      CALL #FW_APW_Oeb_PG
      (  Idx                         := 4 ,
         Niv_Frg                     := #akt_Niv_ZS_AS ,
         Frg_Aus                     := #PW_all_Frg_Aus ,
         Frg_Ein                     := #PW_all_Frg_Ein ,
         DF_Skal                     := 30.0 ,
         IEC_Image                   := "DB_IEC_PW_Image".FW_APW_Oeb_PG ,
         PW_Meld                     := "DB118_PW_Meld".FW_APW_Oeb_PG ,
         PW_Bef                      := "DB119_PW_Bef".FW_APW_Oeb_PG ,
         AS_Zyk                      := #PW_all_Frg_AS_zyk ,
         ZS_Zyk                      := #PW_all_Frg_ZS_zyk ,
         RM_Frg_Ein                  := #PW_all_RM_Frg_Ein ,
         RM_Frg_TeilAus              := #PW_all_RM_Frg_TeilAus ,
         RM_Frg_Aus                  := #PW_all_RM_Frg_Aus
      );

      CALL #FW_APW_Oeb_LW
      (  Idx                         := 5 ,
         Niv_Frg                     := #akt_Niv_ZS_AS ,
         Frg_Aus                     := #PW_all_Frg_Aus ,
         Frg_Ein                     := #PW_all_Frg_Ein ,
         Sperre_ext                  := 0 ,
         DF_Skal                     := 30.0 ,
         IEC_Image                   := "DB_IEC_PW_Image".FW_APW_Oeb_LW ,
         PW_Meld                     := "DB118_PW_Meld".FW_APW_Oeb_LW ,
         PW_Bef                      := "DB119_PW_Bef".FW_APW_Oeb_LW ,
         AS_Zyk                      := #PW_all_Frg_AS_zyk ,
         ZS_Zyk                      := #PW_all_Frg_ZS_zyk ,
         RM_Frg_Ein                  := #PW_all_RM_Frg_Ein ,
         RM_Frg_TeilAus              := #PW_all_RM_Frg_TeilAus ,
         RM_Frg_Aus                  := #PW_all_RM_Frg_Aus
      );

      CALL #FW_APW_GeD_WG
      (  Idx                         := 6 ,
         Niv_Frg                     := #akt_Niv_ZS_AS ,
         Frg_Aus                     := #PW_all_Frg_Aus ,
         Frg_Ein                     := #PW_all_Frg_Ein ,
         IEC_Image                   := "DB_IEC_PW_Image".FW_APW_GeD_WG ,
         PW_Meld                     := "DB118_PW_Meld".FW_APW_GeD_WG ,
         PW_Bef                      := "DB119_PW_Bef".FW_APW_GeD_WG ,
         AS_Zyk                      := #PW_all_Frg_AS_zyk ,
         ZS_Zyk                      := #PW_all_Frg_ZS_zyk ,
         RM_Frg_Ein                  := #PW_all_RM_Frg_Ein ,
         RM_Frg_TeilAus              := #PW_all_RM_Frg_TeilAus ,
         RM_Frg_Aus                  := #PW_all_RM_Frg_Aus
      );

      CALL #FW_APW_GeD_AA
      (  Idx                         := 7 ,
         Niv_Frg                     := #akt_Niv_ZS_AS ,
         Frg_Aus                     := #PW_all_Frg_Aus ,
         Frg_Ein                     := #PW_all_Frg_Ein ,
         IEC_Image                   := "DB_IEC_PW_Image".FW_APW_GeD_AA ,
         PW_Meld                     := "DB118_PW_Meld".FW_APW_GeD_AA ,
         PW_Bef                      := "DB119_PW_Bef".FW_APW_GeD_AA ,
         AS_Zyk                      := #PW_all_Frg_AS_zyk ,
         ZS_Zyk                      := #PW_all_Frg_ZS_zyk ,
         RM_Frg_Ein                  := #PW_all_RM_Frg_Ein ,
         RM_Frg_TeilAus              := #PW_all_RM_Frg_TeilAus ,
         RM_Frg_Aus                  := #PW_all_RM_Frg_Aus
      );

      U "DB118_PW_Meld".FW_APW_WaD.Status.FWA_Betrieb;
      UN #FW_APW_WaD.Sperre_ext;
      S #FW_APW_WeD.Sperre_ext;
      S #FW_APW_NiD.Sperre_ext;

      UN "DB118_PW_Meld".FW_APW_WaD.Status.FWA_Betrieb;
      UN #FW_APW_WaD.Sperre_ext;
      R #FW_APW_WeD.Sperre_ext;
      R #FW_APW_NiD.Sperre_ext;

      CALL #FW_APW_WaD
      (  Idx                         := 8 ,
         Niv_Frg                     := #akt_Niv_ZS_AS ,
         Frg_Aus                     := #PW_all_Frg_Aus ,
         Frg_Ein                     := #PW_all_Frg_Ein ,
         IEC_Image                   := "DB_IEC_PW_Image".FW_APW_WaD ,
         PW_Meld                     := "DB118_PW_Meld".FW_APW_WaD ,
         PW_Bef                      := "DB119_PW_Bef".FW_APW_WaD ,
         AS_Zyk                      := #PW_all_Frg_AS_zyk ,
         ZS_Zyk                      := #PW_all_Frg_ZS_zyk ,
         RM_Frg_Ein                  := #PW_all_RM_Frg_Ein ,
         RM_Frg_TeilAus              := #PW_all_RM_Frg_TeilAus ,
         RM_Frg_Aus                  := #PW_all_RM_Frg_Aus
      );

      U "DB118_PW_Meld".FW_APW_WeD.Status.FWA_Betrieb;
      UN #FW_APW_WeD.Sperre_ext;
      S #FW_APW_WaD.Sperre_ext;
      S #FW_APW_NiD.Sperre_ext;

      UN "DB118_PW_Meld".FW_APW_WeD.Status.FWA_Betrieb;
      UN #FW_APW_WeD.Sperre_ext;
      R #FW_APW_WaD.Sperre_ext;
      R #FW_APW_NiD.Sperre_ext;


      CALL #FW_APW_WeD
      (  Idx                         := 9 ,
         Niv_Frg                     := #akt_Niv_ZS_AS ,
         Frg_Aus                     := #PW_all_Frg_Aus ,
         Frg_Ein                     := #PW_all_Frg_Ein ,
         IEC_Image                   := "DB_IEC_PW_Image".FW_APW_WeD ,
         PW_Meld                     := "DB118_PW_Meld".FW_APW_WeD ,
         PW_Bef                      := "DB119_PW_Bef".FW_APW_WeD ,
         AS_Zyk                      := #PW_all_Frg_AS_zyk ,
         ZS_Zyk                      := #PW_all_Frg_ZS_zyk ,
         RM_Frg_Ein                  := #PW_all_RM_Frg_Ein ,
         RM_Frg_TeilAus              := #PW_all_RM_Frg_TeilAus ,
         RM_Frg_Aus                  := #PW_all_RM_Frg_Aus
      );

      U "DB118_PW_Meld".FW_APW_NiD.Status.FWA_Betrieb;
      UN #FW_APW_NiD.Sperre_ext;
      S #FW_APW_WeD.Sperre_ext;
      S #FW_APW_WaD.Sperre_ext;

      UN "DB118_PW_Meld".FW_APW_NiD.Status.FWA_Betrieb;
      UN #FW_APW_NiD.Sperre_ext;
      R #FW_APW_WeD.Sperre_ext;
      R #FW_APW_WaD.Sperre_ext;

      CALL #FW_APW_NiD
      (  Idx                         := 10 ,
         Niv_Frg                     := #akt_Niv_ZS_AS ,
         Frg_Aus                     := #PW_all_Frg_Aus ,
         Frg_Ein                     := #PW_all_Frg_Ein ,
         IEC_Image                   := "DB_IEC_PW_Image".FW_APW_NiD ,
         PW_Meld                     := "DB118_PW_Meld".FW_APW_NiD ,
         PW_Bef                      := "DB119_PW_Bef".FW_APW_NiD ,
         AS_Zyk                      := #PW_all_Frg_AS_zyk ,
         ZS_Zyk                      := #PW_all_Frg_ZS_zyk ,
         RM_Frg_Ein                  := #PW_all_RM_Frg_Ein ,
         RM_Frg_TeilAus              := #PW_all_RM_Frg_TeilAus ,
         RM_Frg_Aus                  := #PW_all_RM_Frg_Aus
      );

      CALL #FW_APW_LoS
      (  Idx                         := 11 ,
         Niv_Frg                     := #akt_Niv_ZS_AS ,
         Frg_Aus                     := #PW_all_Frg_Aus ,
         Frg_Ein                     := #PW_all_Frg_Ein ,
         IEC_Image                   := "DB_IEC_PW_Image".FW_APW_LoS ,
         PW_Meld                     := "DB118_PW_Meld".FW_APW_LoS ,
         PW_Bef                      := "DB119_PW_Bef".FW_APW_LoS ,
         AS_Zyk                      := #PW_all_Frg_AS_zyk ,
         ZS_Zyk                      := #PW_all_Frg_ZS_zyk ,
         RM_Frg_Ein                  := #PW_all_RM_Frg_Ein ,
         RM_Frg_TeilAus              := #PW_all_RM_Frg_TeilAus ,
         RM_Frg_Aus                  := #PW_all_RM_Frg_Aus
      );

      CALL #FW_APW_Oeb_Ge
      (  Idx                         := 12 ,
         Niv_Frg                     := #akt_Niv_ZS_AS ,
         Frg_Aus                     := #PW_all_Frg_Aus ,
         Frg_Ein                     := #PW_all_Frg_Ein ,
         DF_Skal                     := 20.0 ,
         IEC_Image                   := "DB_IEC_PW_Image".FW_APW_Oeb_Ge ,
         PW_Meld                     := "DB118_PW_Meld".FW_APW_Oeb_Ge ,
         PW_Bef                      := "DB119_PW_Bef".FW_APW_Oeb_Ge ,
         AS_Zyk                      := #PW_all_Frg_AS_zyk ,
         ZS_Zyk                      := #PW_all_Frg_ZS_zyk ,
         RM_Frg_Ein                  := #PW_all_RM_Frg_Ein ,
         RM_Frg_TeilAus              := #PW_all_RM_Frg_TeilAus ,
         RM_Frg_Aus                  := #PW_all_RM_Frg_Aus
      );

      CALL #FW_APW_BuH
      (  Idx                         := 13 ,
         Niv_Frg                     := #akt_Niv_ZS_AS ,
         Frg_Aus                     := #PW_all_Frg_Aus ,
         Frg_Ein                     := #PW_all_Frg_Ein ,
         IEC_Image                   := "DB_IEC_PW_Image".FW_APW_BuH ,
         PW_Meld                     := "DB118_PW_Meld".FW_APW_BuH ,
         PW_Bef                      := "DB119_PW_Bef".FW_APW_BuH ,
         AS_Zyk                      := #PW_all_Frg_AS_zyk ,
         ZS_Zyk                      := #PW_all_Frg_ZS_zyk ,
         RM_Frg_Ein                  := #PW_all_RM_Frg_Ein ,
         RM_Frg_TeilAus              := #PW_all_RM_Frg_TeilAus ,
         RM_Frg_Aus                  := #PW_all_RM_Frg_Aus
      );

      CALL #FW_APW_BrR_TS
      (  Idx                         := 14 ,
         Niv_Frg                     := #akt_Niv_ZS_AS ,
         Frg_Aus                     := #PW_all_Frg_Aus ,
         Frg_Ein                     := #PW_all_Frg_Ein ,
         IEC_Image                   := "DB_IEC_PW_Image".FW_APW_BrR_TS ,
         PW_Meld                     := "DB118_PW_Meld".FW_APW_BrR_TS ,
         PW_Bef                      := "DB119_PW_Bef".FW_APW_BrR_TS ,
         AS_Zyk                      := #PW_all_Frg_AS_zyk ,
         ZS_Zyk                      := #PW_all_Frg_ZS_zyk ,
         RM_Frg_Ein                  := #PW_all_RM_Frg_Ein ,
         RM_Frg_TeilAus              := #PW_all_RM_Frg_TeilAus ,
         RM_Frg_Aus                  := #PW_all_RM_Frg_Aus
      );

NETWORK
TITLE = Steuerung Zulauf/Freigabe Pumpwerke - Status - alle Freigaben
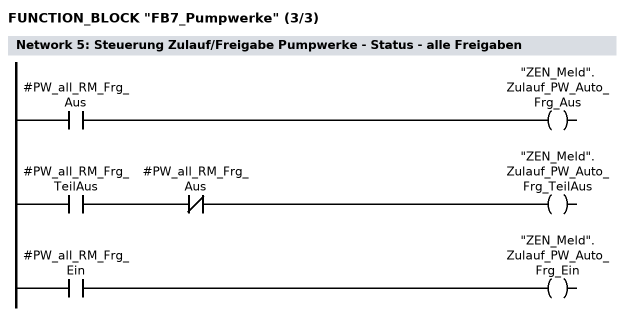

      U #PW_all_RM_Frg_Aus;
      = "ZEN_Meld".Zulauf_PW_Auto_Frg_Aus;
      U #PW_all_RM_Frg_TeilAus;
      UN #PW_all_RM_Frg_Aus;
      = "ZEN_Meld".Zulauf_PW_Auto_Frg_TeilAus;
      U #PW_all_RM_Frg_Ein;
      = "ZEN_Meld".Zulauf_PW_Auto_Frg_Ein;


END_FUNCTION_BLOCK

FUNCTION_BLOCK "FB8_Leitstelle"
{ S7_Optimized_Access := 'TRUE' }
VERSION : 0.1
   VAR_TEMP
      BB_G1_SS : Bool;
      BB_G2_SS : Bool;
      BB_G3_SS : Bool;
      retval : Int;
   END_VAR


BEGIN
NETWORK
TITLE = Sammelmeldung an Leitstelle - Gebläse 1 Störung
      U "DB104_Antriebe_Meld".BB_G1.Status.BB_SS;
      O "DB104_Antriebe_Meld".BB_G1.Stoerung.St_Kom_DP;
      = #BB_G1_SS;
      U "DB104_Antriebe_Meld".BB_G2.Status.BB_SS;
      O "DB104_Antriebe_Meld".BB_G2.Stoerung.St_Kom_DP;
      = #BB_G2_SS;
      U "DB104_Antriebe_Meld".BB_G3.Status.BB_SS;
      O "DB104_Antriebe_Meld".BB_G3.Stoerung.St_Kom_DP;
      = #BB_G3_SS;

//Gebläse 1 Störung
      U #BB_G1_SS;
      = "ZEN_Meld".IEC_Meld_LS_001;
//Gebläse 2 Störung
      U #BB_G2_SS;
      = "ZEN_Meld".IEC_Meld_LS_002;
//Gebläse 3 Störung
      U #BB_G3_SS;
      = "ZEN_Meld".IEC_Meld_LS_003;

//Belebungsbecken 1 Rezipumpe 1 Störung
      U "DB104_Antriebe_Meld".BB1_RZP1.Status.BB_SS;
      = "ZEN_Meld".IEC_Meld_LS_004;

//Belebungsbecken 1 Rezipumpe 2 Störung
      U "DB104_Antriebe_Meld".BB1_RZP2.Status.BB_SS;
      = "ZEN_Meld".IEC_Meld_LS_005;

//Belebungsbecken 1 Überschussschlammpumpe Störung
      U "DB104_Antriebe_Meld".BB1_UeSP.Status.BB_SS;
      = "ZEN_Meld".IEC_Meld_LS_006;

//Belebungsbecken 1 Ablaufschieber Störung
      U "DB104_Antriebe_Meld".BB1_AS1.Status.BB_SS;
      O "DB104_Antriebe_Meld".BB1_AS2.Status.BB_SS;
      = "ZEN_Meld".IEC_Meld_LS_007;

//Belebungsbecken 1 Schlammrückführung Störung
      U "DB104_Antriebe_Meld".BB1_SR1.Status.BB_SS;
      O "DB104_Antriebe_Meld".BB1_SR2.Status.BB_SS;
      = "ZEN_Meld".IEC_Meld_LS_008;

//Belebungsbecken 2 Rezipumpe 1 Störung
      U "DB104_Antriebe_Meld".BB2_RZP1.Status.BB_SS;
      = "ZEN_Meld".IEC_Meld_LS_009;

//Belebungsbecken 2 Rezipumpe 2 Störung
      U "DB104_Antriebe_Meld".BB2_RZP2.Status.BB_SS;
      = "ZEN_Meld".IEC_Meld_LS_010;

//Belebungsbecken 2 Überschussschlammpumpe Störung
      U "DB104_Antriebe_Meld".BB2_UeSP.Status.BB_SS;
      = "ZEN_Meld".IEC_Meld_LS_011;

//Belebungsbecken 2 Ablaufschieber Störung
      U "DB104_Antriebe_Meld".BB2_AS1.Status.BB_SS;
      O "DB104_Antriebe_Meld".BB2_AS2.Status.BB_SS;
      = "ZEN_Meld".IEC_Meld_LS_012;

//Belebungsbecken 2 Schlammrückführung Störung
      U "DB104_Antriebe_Meld".BB2_SR1.Status.BB_SS;
      O "DB104_Antriebe_Meld".BB2_SR2.Status.BB_SS;
      = "ZEN_Meld".IEC_Meld_LS_013;

//Rechenanlage Störung
      U "DB104_Antriebe_Meld".Zulauf_RA_FP.Status.BB_SS;
      O "DB104_Antriebe_Meld".Zulauf_RA_SA.Status.BB_SSnq;
      O "DB104_Antriebe_Meld".Zulauf_RA_HZS.Status.BB_SS;
      O "DB104_Antriebe_Meld".Zulauf_RA_VKS.Status.BB_SS;
      O "DB104_Antriebe_Meld".Zulauf_RA_V.Status.BB_SS;
      O "DB104_Antriebe_Meld".Zulauf_RA_RP.Status.BB_SS;
      = "ZEN_Meld".IEC_Meld_LS_014;

//Schlammpumpe Störung
      U "DB104_Antriebe_Meld".Schlamm_BP.Status.BB_SS;
      = "ZEN_Meld".IEC_Meld_LS_015;

//Eindicker Störung
      CLR;
      = "ZEN_Meld".IEC_Meld_LS_016;

//Trübwasserpumpe Störung
      U "DB104_Antriebe_Meld".Truebwasser_P1.Status.BB_SS;
      O "DB104_Antriebe_Meld".Truebwasser_P2.Status.BB_SS;
      = "ZEN_Meld".IEC_Meld_LS_017;

//Schlammstapelbehälter Störung
      U "DB104_Antriebe_Meld".Schlamm_AS.Status.BB_SS;
      = "ZEN_Meld".IEC_Meld_LS_018;

//Druckluftkompressor Störung
      U "DB104_Antriebe_Meld".BB1_SR_K.Status.BB_SS;
      O "DB104_Antriebe_Meld".BB2_SR_K.Status.BB_SS;
      = "ZEN_Meld".IEC_Meld_LS_019;

//Zulaufschieber Störung
      U "DB104_Antriebe_Meld".Zulauf_AS.Status.BB_SS;
      = "ZEN_Meld".IEC_Meld_LS_020;

//Luftschieber Störung
      U "DB104_Antriebe_Meld".BB_LS1.Status.BB_SS;
      O "DB104_Antriebe_Meld".BB_LS2.Status.BB_SS;
      = "ZEN_Meld".IEC_Meld_LS_021;

//Filtration Störung
      CLR;
      = "ZEN_Meld".IEC_Meld_LS_022;
//Reserve 23
      = "ZEN_Meld".IEC_Meld_LS_023;
//Netzausfall
      O "ZEN_Meld".E_NSHV_NA;
      O "ZEN_Meld".SimpleSignalingStatus_BF_Bit00;
      O "ZEN_Meld".SimpleSignalingStatus_BF_Bit01;
      = "ZEN_Meld".IEC_Meld_LS_024;

//400VAC/24VDC Sammelstörung
      U "ZEN_Meld".E_NSHV_SS1_St;
      O "ZEN_Meld".E_NSHV_SS2_St;
      O "ZEN_Meld".E_NSHV_N02_AF_St;
      O "ZEN_Meld".E_NSHV_N03_AF_St;
      O "ZEN_Meld".E_NSHV_N04_AF_St;
      O "ZEN_Meld".E_NSHV_LS_Aus;
      O "ZEN_Meld".E_NSHV_LS_St;
      = "ZEN_Meld".IEC_Meld_LS_025;

//Mengenmessung Störung
      U "DB114_MW_Meld".Zulauf_AR_DF.Status.BB_SS;
      O "DB114_MW_Meld".Ablauf_DF.Status.BB_SS;
      O "DB114_MW_Meld".Zulauf_DF.Status.BB_SS;
      O "DB114_MW_Meld".BB_UeSS_DF.Status.BB_SS;
      O "DB114_MW_Meld".Schlamm_Besch_DF.Status.BB_SS;
      O "DB114_MW_Meld".Truebwasser_DF.Status.BB_SS;
      = "ZEN_Meld".IEC_Meld_LS_026;

//Biologie Sammelstörung
      U #BB_G1_SS;
      U #BB_G2_SS;
      O(;
      U #BB_G1_SS;
      U #BB_G3_SS;
      );
      O(;
      U #BB_G2_SS;
      U #BB_G3_SS;
      );

      O "ZEN_Meld".E_BB_RT;
      = "ZEN_Meld".IEC_Meld_LS_027;

//Belebungsbecken 1 Biologie Störung
      U "DB114_MW_Meld".BB1_O2.Stoerung.GW_LL;
      O "DB114_MW_Meld".BB1_O2.Status.BB_SS;
      = "ZEN_Meld".IEC_Meld_LS_028;

//Belebungsbecken 2 Biologie Störung
      U "DB114_MW_Meld".BB2_O2.Stoerung.GW_LL;
      O "DB114_MW_Meld".BB2_O2.Status.BB_SS;
      = "ZEN_Meld".IEC_Meld_LS_029;

//Höhenstände Pumpwerke Störung
      U "DB118_PW_Meld".FW_APW_Oeb_KB.Status.MW_Niv_St;
      O "DB118_PW_Meld".FW_APW_BrR_DM.Status.MW_Niv_St;
//      O     "DB118_PW_Meld".FW_APW_Oeb_Tu.Status.MW_Niv_St
      O "DB118_PW_Meld".FW_APW_Oeb_KS.Status.MW_Niv_St;
      O "DB118_PW_Meld".FW_APW_Oeb_PG.Status.MW_Niv_St;
      O "DB118_PW_Meld".FW_APW_Oeb_LW.Status.MW_Niv_St;
      O "DB118_PW_Meld".FW_APW_GeD_WG.Status.MW_Niv_St;
      O "DB118_PW_Meld".FW_APW_GeD_AA.Status.MW_Niv_St;
      O "DB118_PW_Meld".FW_APW_WaD.Status.MW_Niv_St;
      O "DB118_PW_Meld".FW_APW_WeD.Status.MW_Niv_St;
      O "DB118_PW_Meld".FW_APW_NiD.Status.MW_Niv_St;
      O "DB118_PW_Meld".FW_APW_LoS.Status.MW_Niv_St;
      O "DB118_PW_Meld".FW_APW_Oeb_Ge.Status.MW_Niv_St;
      O "DB118_PW_Meld".FW_APW_BuH.Status.MW_Niv_St;
      O "DB118_PW_Meld".FW_APW_BrR_TS.Status.MW_Niv_St;
      = "ZEN_Meld".IEC_Meld_LS_030;

//Höhenstände Kläranlage Störung
      U "DB114_MW_Meld".Zulauf_AR_Niv.Status.BB_SS;
      O "DB114_MW_Meld".Zulauf_AR_Niv.Stoerung.GW_HH;
      O "ZEN_Meld".E_Zulauf_AR_HW;
      O "DB114_MW_Meld".Zulauf_Niv.Status.BB_SS;
      O "DB114_MW_Meld".Zulauf_Niv.Stoerung.GW_HH;
      O "DB114_MW_Meld".Truebwasser_Niv.Status.BB_SS;
      O "DB114_MW_Meld".Truebwasser_Niv.Stoerung.GW_HH;
      = "ZEN_Meld".IEC_Meld_LS_031;

//Türkontakt/Alarmanlage
      U "ZEN_Meld".ZEN_ObjS_Alarm;
      = "ZEN_Meld".IEC_Meld_LS_032;

NETWORK
TITLE = Messwerte Wetterstation

      L "DB114_MW_Meld".Umwelt_WG.MW_akt;
      L 0.0;
      <R;
      SPB WGzw;
      TAK;
WGzw:      T "DB_IEC_MW_Image".Umwelt_WG.Data_TK36;
      L "DB114_MW_Meld".Umwelt_WR.MW_akt;
      L 0.0;
      <R;
      SPB WRzw;
      TAK;
      L 360.0;
      >R;
      SPB WRzw;
      TAK;
WRzw:      T "DB_IEC_MW_Image".Umwelt_WR.Data_TK36;
      L "DB114_MW_Meld".Umwelt_LDr.MW_akt;
      T "DB_IEC_MW_Image".Umwelt_LDr.Data_TK36;
      L "DB114_MW_Meld".Umwelt_T.MW_akt;
      T "DB_IEC_MW_Image".Umwelt_T.Data_TK36;
      L "DB114_MW_Meld".Umwelt_LF.MW_akt;
      T "DB_IEC_MW_Image".Umwelt_LF.Data_TK36;

      U "DB114_MW_Meld".Umwelt_WG.Status.BB_SS;
      CLR;
      = "DB_IEC_MW_Image".Umwelt_WG.IV;
      U "DB114_MW_Meld".Umwelt_WR.Status.BB_SS;
      CLR;
      = "DB_IEC_MW_Image".Umwelt_WR.IV;
      U "DB114_MW_Meld".Umwelt_LDr.Status.BB_SS;
      = "DB_IEC_MW_Image".Umwelt_LDr.IV;
      U "DB114_MW_Meld".Umwelt_T.Status.BB_SS;
      = "DB_IEC_MW_Image".Umwelt_T.IV;
      U "DB114_MW_Meld".Umwelt_LF.Status.BB_SS;
      = "DB_IEC_MW_Image".Umwelt_LF.IV;

      L "ZEN_MW".Umwelt_RM_ZW;
      RND;
      T "DB_IEC_MW_Image".Umwelt_RM.Data_TK37;




      CALL RD_LOC_T
      {date_type := 'Date_And_Time'}
      (  RET_VAL                     := #retval ,
         OUT                         := "DB_IEC_MW_Image".Umwelt_RM.TS
      );
END_FUNCTION_BLOCK

FUNCTION_BLOCK "FB9_USV_Kom"
{ S7_Optimized_Access := 'TRUE' }
VERSION : 0.1
   VAR
      TSEND_Instance {InstructionName := 'TSEND'; LibVersion := '4.0'} : TSEND;
      TRCV_Instance {InstructionName := 'TRCV'; LibVersion := '4.0'} : TRCV;
      USV_MB : "FB78_ModbusOverIP_USV";
      Send_Req { S7_SetPoint := 'True'} : Bool;
      Send_Done : Bool;
      Send_Busy : Bool;
      Send_Error : Bool;
      Rec_NDR : Bool;
      Rec_Busy : Bool;
      Rec_Error : Bool;
      cmd_aux1 : Bool;
      cmd_aux2 : Bool;
      Send_Status : Word;
      Rec_Status : Word;
      Send_Len : UDInt;
      Rec_Len : UDInt;
   END_VAR

   VAR_TEMP
      retval : Int;
      tmp_DI : DInt;
   END_VAR


BEGIN
NETWORK
TITLE =


      CALL #TSEND_Instance
      {data_type := 'Variant', len_type := 'UDInt', id_type := 'CONN_OUC'}
      (  REQ                         := #Send_Req ,
         ID                          := 16#100 ,
         LEN                         := #Send_Len ,
         DONE                        := #Send_Done ,
         BUSY                        := #Send_Busy ,
         ERROR                       := #Send_Error ,
         STATUS                      := #Send_Status ,
         DATA                        := "DB60_USV_ModTCP_SEND".Data
      );

      CALL #TRCV_Instance
      {ptr_type := 'Variant', value_type := 'UDInt', id_type := 'CONN_OUC'}
      (  EN_R                        := 1 ,
         ID                          := 16#100 ,
         LEN                         := 0 ,
         ADHOC                       := 1 ,
         NDR                         := #Rec_NDR ,
         BUSY                        := #Rec_Busy ,
         ERROR                       := #Rec_Error ,
         STATUS                      := #Rec_Status ,
         RCVD_LEN                    := #Rec_Len ,
         DATA                        := "DB59_USV_ModTCP_RCV".Data
      );


      CALL #USV_MB
      (  Rec_ok                      := #Rec_NDR ,
         Send_ok                     := #Send_Done ,
         Rec_Len                     := #Rec_Len ,
         Send_Req                    := #Send_Req ,
         Kom_St                      := "ZEN_Meld".UPSStatus_SF_Msg08 ,
         Send_Len                    := #Send_Len ,
         Cmd_Aux01                   := #cmd_aux1 ,
         Cmd_Aux02                   := #cmd_aux2
      );

NETWORK
TITLE = Zuweisungen auf Melde-DBs

      CALL "FC41_Modbus2Proc_DI"
      (  ModReg                      := "DB61_USV_ModTCP_WorkData".REQ02.Reg128 ,
         Faktor                      := 1.0 ,
         enable                      := 1 ,
         Value                       := "ZEN_MW".RunTimeRemaining
      );

      L "DB61_USV_ModTCP_WorkData".REQ02.Reg130;
      T #tmp_DI;

      CALL "FC41_Modbus2Proc_DI"
      (  ModReg                      := #tmp_DI ,
         Faktor                      := 0.001953125 ,
         enable                      := 1 ,
         Value                       := "ZEN_MW".StateOfCharge_Pct
      );



//Meldungen

      L "DB61_USV_ModTCP_WorkData".REQ01.Reg000_l;
      T %DB100.DBW168;
      L "DB61_USV_ModTCP_WorkData".REQ01.Reg000_h;
      T %DB100.DBW166;
      L "DB61_USV_ModTCP_WorkData".REQ01.Reg018;
      T %DB100.DBW170;

      L "DB61_USV_ModTCP_WorkData".REQ01.Reg019;
      L 0;
      <>I;
      = "ZEN_Meld".UPSStatus_SF_Msg01;
      L "DB61_USV_ModTCP_WorkData".REQ01.Reg020;
      L DINT#0;
      <>D;
      = "ZEN_Meld".UPSStatus_SF_Msg02;
      L "DB61_USV_ModTCP_WorkData".REQ01.Reg022;
      L 0;
      <>I;
      = "ZEN_Meld".UPSStatus_SF_Msg03;


END_FUNCTION_BLOCK

ORGANIZATION_BLOCK "Pull or plug of modules"
{ S7_Optimized_Access := 'TRUE' }
VERSION : 0.1

BEGIN
NETWORK
TITLE =
END_ORGANIZATION_BLOCK

ORGANIZATION_BLOCK "Rack or station failure"
{ S7_Optimized_Access := 'TRUE' }
VERSION : 0.1

BEGIN
NETWORK
TITLE =
END_ORGANIZATION_BLOCK

ORGANIZATION_BLOCK "Programming error"
{ S7_Optimized_Access := 'TRUE' }
VERSION : 0.1

BEGIN
NETWORK
TITLE =
END_ORGANIZATION_BLOCK

FUNCTION "FC40_Modbus2Proc" : Void
{ S7_Optimized_Access := 'TRUE' }
VERSION : 0.1
   VAR_INPUT
      ModReg : Int;
      Faktor : Real;
      enable : Bool;
   END_VAR

   VAR_IN_OUT
      Value : Real;
   END_VAR


BEGIN
NETWORK
TITLE =
      UN #enable;
      BEB;

      L #ModReg;
      ITD;
      DTR;
      L #Faktor;
      *R;
      T #Value;

END_FUNCTION

